// Implicitly generated code : DO NOT EDIT
FUNCTION CheckRangeUnsigned : UDINT
VAR_INPUT
	value, lower, upper: UDINT;
END_VAR

// Implicitly generated code: Only an implementation suggestion
{noflow}
IF (value < lower) THEN
	CheckRangeUnsigned := lower;
ELSIF(value > upper) THEN
	CheckRangeUnsigned := upper;
ELSE
	CheckRangeUnsigned := value;
END_IF

END_FUNCTION

(* stored: Version 1.1.0.1
   POU CheckRangeUnsigned: Id {ec2d47fe-8ca9-4778-b683-143c269b566e}, SpecialFunc CheckRangeUnsigned *)
